// TIA Portal V19 export
VAR_GLOBAL   // PLC tag table "TT - Reject"
   iRejectSenCilIn_f0 AT %I1.1 : Bool;
   iRejectSenCilOut_f1 AT %I1.2 : Bool;
   iRejectSenCilUp_g0 AT %I1.3 : Bool;
   "oRejectVenCilOut_F+" AT %Q0.6 : Bool;   // Bistabiel
   "oRejectVenCilIn_F-" AT %Q0.7 : Bool;   // Bistabiel
   oRejectVenCilDown_E AT %Q1.0 : Bool;
   "oRejectVenVacuum_V+" AT %Q1.1 : Bool;
   "iRejectSenVacuum_V+" AT %I2.1 : Bool;   // true when vacuum
END_VAR
